FUNCTION BOOL_TO_DINT : DINT
	VAR_INPUT
		in : BOOL;
	END_VAR
BEGIN
	IF in = true THEN
		BOOL_TO_DINT := 1 ;
	ELSE
		BOOL_TO_DINT := 0 ;
	END_IF ;
END_FUNCTION